INTERFACE I_RpcHandlers

METHOD PUBLIC RegisterHandler
VAR_INPUT
	MethodName : T_MAXSTRING;
	Handler : I_RpcHandler;
END_VAR
END_METHOD

METHOD PUBLIC TryGetByMethodName : BOOL
VAR_INPUT
	MethodName : T_MAXSTRING;
	Destination : REFERENCE TO I_RpcHandler;
END_VAR
END_METHOD

END_INTERFACE

(* stored: Version 1.1.0.1, ProductVersion 3.1.4024.12
   Itf I_RpcHandlers: Id {d33e8c48-0ad7-4d08-bfcf-6104e8ce9bf4}
   Method RegisterHandler: Id {b3ef9631-08be-494d-b8c5-fe3c03e037ec}
   Method TryGetByMethodName: Id {7dcc2284-1e0a-4e94-8249-d87a74da0f15} *)
